PROGRAM P_WinchControl
VAR
END_VAR

END_PROGRAM

(* stored: Version 1.1.0.1, ProductVersion 3.1.4024.11
   POU P_WinchControl: Id {9db37c6e-a65f-4d33-b11a-5f984ef248b2}, SpecialFunc None *)
